FUNCTION FC_MarkingLayoutSelection : STRING(243)
VAR_INPUT
	Source	: eMarkingLayoutSource;
	Text	: STRING;
	MarkingCode : STRING(243);
	ProductName : STRING(243);
END_VAR

IF Source = eMarkingLayoutSource.ProductName THEN
	FC_MarkingLayoutSelection := ProductName;
ELSIF Source = eMarkingLayoutSource.FreeText THEN
	FC_MarkingLayoutSelection := Text;
ELSE
	FC_MarkingLayoutSelection := MarkingCode;
END_IF

END_FUNCTION

(* stored: Version 1.1.0.1, ProductVersion 3.1.4024.13
   POU FC_MarkingLayoutSelection: Id {90d0128c-a569-4c4c-99da-e31172dadb45}, SpecialFunc None *)
